INTERFACE IStringContainer EXTENDS IHaveValue

PROPERTY text : STRING(255)
GET
END_GET
SET
END_SET
END_PROPERTY

END_INTERFACE

(* stored: Version 1.1.0.1
   Itf IStringContainer: Id {5a8f6dc7-6a29-4589-82b3-8496910bf3df}
   Property text: Id {c68aa7aa-f694-4617-b547-2d74ea10483b}
   Get Get: Id {9cbd87cb-335a-4d0e-9626-1633ebf9d259}
   Set Set: Id {ee4feb52-11c5-4b80-a690-8a8c40d29d6b} *)
